INTERFACE I_DataChannelRecv

PROPERTY Error : INT
GET
END_GET
SET
END_SET
END_PROPERTY

PROPERTY DataSize : UDINT
GET
END_GET
END_PROPERTY

PROPERTY Busy : BOOL
GET
END_GET
END_PROPERTY

{attribute 'object_name' := 'InitChannel'}
METHOD InitChannel : BOOL
VAR_INPUT
	udiDataSize: UDINT;
	pInputData: POINTER TO BYTE;
END_VAR
END_METHOD

{attribute 'object_name' := 'GetData'}
METHOD GetData : BOOL
VAR_INPUT
	udiDataSize: UDINT;
	pData: POINTER TO BYTE;
END_VAR
END_METHOD

END_INTERFACE

(* stored: Version 1.1.0.1, ProductVersion 3.1.0.26
   Itf I_DataChannelRecv: Id {e5eaf0da-b144-4e0f-9d32-d5071ca5335e}
   Property Error: Id {0372085c-546d-40c4-9201-4ba569e31b85}
   Get Get: Id {3dbe34ba-fd92-4c63-8779-8730611d7302}
   Set Set: Id {90818e4f-13c3-4b6d-85f1-5f17bc47c651}
   Property DataSize: Id {1a1bf648-56b6-46f7-a876-3db2727e3b62}
   Get Get: Id {c2b9a4c9-675d-46b6-849f-ac993f4e3d07}
   Property Busy: Id {66cbc28e-689c-422f-8935-4657a26bda89}
   Get Get: Id {185ed716-6d07-4c80-8d5d-19aadf41c4dd}
   Method InitChannel: Id {7f351c00-5711-4536-af78-61e36b5f7fbe}
   Method GetData: Id {cee20ce2-704f-4bf3-93bd-983ae446da25} *)
